INTERFACE I_Diagnosable

PROPERTY ErrorId : UDINT
GET
END_GET
END_PROPERTY

END_INTERFACE

(* stored: Version 1.1.0.1, ProductVersion 3.1.4024.12
   Itf I_Diagnosable: Id {44f24c7f-e41c-459d-bbef-03726f4cb7f7}
   Property ErrorId: Id {1d33b91d-7479-4e10-b98e-7913ca5214a4}
   Get Get: Id {09629565-e2b2-4ba6-914c-8ce06412ee33} *)
